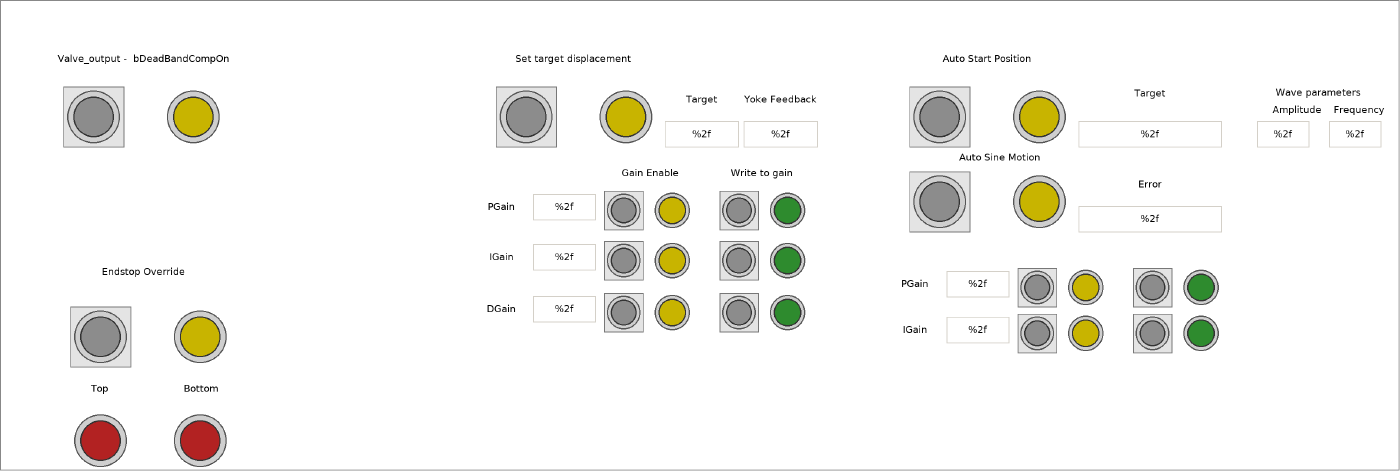
VISUALIZATION Engineer_HMI  // 1615x544
    PushSwitch (73,100 70x70), variable: G_Parameters.stParam.bWinchDeadBandCompOn, behaviour: TOGGLE, style: Switch-PushSwitch-Gray
    Lamp1 (188,100 70x70), variable: G_Parameters.stParam.bWinchDeadBandCompOn, style: Lamp-Lamp1-Yellow
    Label (33,53 265x30), "Valve_output - bDeadBandCompOn"
    PushSwitch (81,354 70x70), variable: G_Engineer_HMI.bEndStopOverride, behaviour: TOGGLE, style: Switch-PushSwitch-Gray
    Lamp1 (196,354 70x70), variable: G_Engineer_HMI.bEndStopOverride, style: Lamp-Lamp1-Yellow
    Label (33,299 265x30), "Endstop Override"
    Lamp1 (81,474 70x70), variable: G_Engineer_HMI.bEndStopUpActive, style: Lamp-Lamp1-Red
    Lamp1 (196,474 70x70), variable: G_Engineer_HMI.bEndStopDownActive, style: Lamp-Lamp1-Red
    Label (81,434 68x30), "Top"
    Label (198,434 68x30), "Bottom"
    PushSwitch (572,100 70x70), variable: G_Engineer_HMI.bDisplacement_target_active, behaviour: TOGGLE, style: Switch-PushSwitch-Gray
    Lamp1 (687,100 70x70), variable: G_Engineer_HMI.bDisplacement_target_active, style: Lamp-Lamp1-Yellow
    Label (767,100 85x30), "Target"
    Label (557,224 43x30), "PGain"
    Label (557,53 209x30), "Set target displacement"
    Textfield (767,140 85x30), "%2f", text variable: G_Engineer_HMI.fDisplacement_target
        OnMouseClick: write G_Engineer_HMI.fDisplacement_target via Default
    PushSwitch (697,218 45x50), variable: G_Engineer_HMI.bPenable_dis, behaviour: TOGGLE, style: Switch-PushSwitch-Gray
    Lamp1 (752,218 47x50), variable: G_Engineer_HMI.bPenable_dis, style: Lamp-Lamp1-Yellow
    Textfield (615,224 72x30), "%2f", text variable: G_Engineer_HMI.fProportionalgain_dis
        OnMouseClick: write G_Engineer_HMI.fProportionalgain_dis via Default
    Label (830,185 98x30), "Write to gain"
    Label (701,185 98x30), "Gain Enable"
    PushSwitch (830,218 45x50), variable: G_Engineer_HMI.bPenable_dis_write, behaviour: TOGGLE, style: Switch-PushSwitch-Gray
    Lamp1 (885,218 47x50), variable: G_Engineer_HMI.bPenable_dis_write, style: Lamp-Lamp1-Green
    Label (557,282 43x30), "IGain"
    PushSwitch (697,276 45x50), variable: G_Engineer_HMI.bIenable_dis, behaviour: TOGGLE, style: Switch-PushSwitch-Gray
    Lamp1 (752,276 47x50), variable: G_Engineer_HMI.bIenable_dis, style: Lamp-Lamp1-Yellow
    Textfield (615,282 72x30), "%2f", text variable: G_Engineer_HMI.fIntegralgain_dis
        OnMouseClick: write G_Engineer_HMI.fIntegralgain_dis via Default
    PushSwitch (830,276 45x50), variable: G_Engineer_HMI.bIenable_dis_write, behaviour: TOGGLE, style: Switch-PushSwitch-Gray
    Lamp1 (885,276 47x50), variable: G_Engineer_HMI.bIenable_dis_write, style: Lamp-Lamp1-Green
    Label (557,342 43x30), "DGain"
    PushSwitch (697,336 45x50), variable: G_Engineer_HMI.bDenable_dis, behaviour: TOGGLE, style: Switch-PushSwitch-Gray
    Lamp1 (752,336 47x50), variable: G_Engineer_HMI.bDenable_dis, style: Lamp-Lamp1-Yellow
    Textfield (615,342 72x30), "%2f", text variable: G_Engineer_HMI.fDerivativegain_dis
        OnMouseClick: write G_Engineer_HMI.fDerivativegain_dis via Default
    PushSwitch (830,336 45x50), variable: G_Engineer_HMI.bDenable_dis_write, behaviour: TOGGLE, style: Switch-PushSwitch-Gray
    Lamp1 (885,336 47x50), variable: G_Engineer_HMI.bDenable_dis_write, style: Lamp-Lamp1-Green
    PushSwitch (1049,100 70x70), variable: G_Engineer_HMI.bAutoStartPosEnable, behaviour: TOGGLE, style: Switch-PushSwitch-Gray
    Lamp1 (1164,100 70x70), variable: G_Engineer_HMI.bAutoStartPosEnable, style: Lamp-Lamp1-Yellow
    Label (1034,53 209x30), "Auto Start Position"
    Textfield (1244,140 165x30), "%2f", text variable: G_Engineer_HMI.fAutoStartPos_target
        OnMouseClick: write G_Engineer_HMI.fAutoStartPos_target via Default
    Label (1034,313 43x30), "PGain"
    PushSwitch (1174,307 45x50), variable: G_Engineer_HMI.bPenable_MOOG, behaviour: TOGGLE, style: Switch-PushSwitch-Gray
    Lamp1 (1229,307 47x50), variable: G_Engineer_HMI.bPenable_MOOG, style: Lamp-Lamp1-Yellow
    Textfield (1092,313 72x30), "%2f", text variable: G_Engineer_HMI.fProportionalgain_MOOG
        OnMouseClick: write G_Engineer_HMI.fProportionalgain_MOOG via Default
    PushSwitch (1307,307 45x50), variable: G_Engineer_HMI.bPenable_MOOG_write, behaviour: TOGGLE, style: Switch-PushSwitch-Gray
    Lamp1 (1362,307 47x50), variable: G_Engineer_HMI.bPenable_MOOG_write, style: Lamp-Lamp1-Green
    PushSwitch (1049,198 70x70), variable: G_Engineer_HMI.bAutoSineMotionEnable, behaviour: TOGGLE, style: Switch-PushSwitch-Gray
    Lamp1 (1164,198 70x70), variable: G_Engineer_HMI.bAutoSineMotionEnable, style: Lamp-Lamp1-Yellow
    Label (1049,167 209x30), "Auto Sine Motion"
    Textfield (1244,238 165x30), "%2f", text variable: G_Motion_Control.fPosition_error_SineMotion
    Label (1034,366 43x30), "IGain"
    PushSwitch (1174,360 45x50), variable: G_Engineer_HMI.bIenable_MOOG, behaviour: TOGGLE, style: Switch-PushSwitch-Gray
    Lamp1 (1229,360 47x50), variable: G_Engineer_HMI.bIenable_MOOG, style: Lamp-Lamp1-Yellow
    Textfield (1092,366 72x30), "%2f", text variable: G_Engineer_HMI.fIntegrationalgain_MOOG
        OnMouseClick: write G_Engineer_HMI.fIntegrationalgain_MOOG via Default
    PushSwitch (1307,360 45x50), variable: G_Engineer_HMI.bIenable_MOOG_write, behaviour: TOGGLE, style: Switch-PushSwitch-Gray
    Lamp1 (1362,360 47x50), variable: G_Engineer_HMI.bIenable_MOOG_write, style: Lamp-Lamp1-Green
    Label (1244,93 165x30), "Target"
    Label (1244,198 165x30), "Error"
    Label (1438,92 165x30), "Wave parameters"
    Textfield (1450,140 60x30), "%2f", text variable: G_Engineer_HMI.fAmp
        OnMouseClick: write G_Engineer_HMI.fAmp via Default
    Textfield (1533,140 60x30), "%2f", text variable: G_Engineer_HMI.fFreq
        OnMouseClick: write G_Engineer_HMI.fFreq via Default
    Label (1450,112 165x30), "Amplitude Frequency"
    Label (858,100 85x30), "Yoke Feedback"
    Textfield (858,140 85x30), "%2f", text variable: G_Sensors.fYokeNormalizedFeedback
END_VISUALIZATION

(* stored: Version 1.1.0.1
   Visu Engineer_HMI: Id {3c046ea6-2ad7-430d-94b1-38b7ccc8e80e} *)
